{attribute 'GeneratedUsingTerminal: EL5101-0000-1020'}
{attribute addProperty BoxType "EL5101-0000-1020"}
{attribute addProperty Id "ControlAT %Q*Control_6EF2C5D04Set_counter_valueAT %Q*UINT2"}
{attribute addProperty CRC "568512845"}
{attribute addProperty Size "6"}
TYPE ENC_Control_compact_21E2D14D :
STRUCT
	{attribute addProperty Name "Control"}
	Control AT %Q* : Control_6EF2C5D0;
	{attribute addProperty Name "Set_counter_value"}
	Set_counter_value AT %Q* : UINT;
END_STRUCT
END_TYPE

(* stored: Version 1.2.0.0, ProductVersion 3.1.4024.9
   DUT ENC_Control_compact_21E2D14D: Id {29d0e0bd-76eb-4a4e-a079-985f1ec2de87} *)
